// TIA Portal V20 export
TYPE "LER_typeServoTorqueCalConfigruation"
// stored: Access Published
   STRUCT
      Alarm_Disable : Bool;
      OverLoad_Warning_SV : LReal;
      OverLoad_Alarm_SV : LReal;
   END_STRUCT;
END_TYPE
